INTERFACE ITF_BaseControlElement_HMI_Connector_Command

END_INTERFACE

(* stored: Version 1.1.0.1
   Itf ITF_BaseControlElement_HMI_Connector_Command: Id {78690def-5583-0bf8-09a4-f698b1eeeb2d} *)
